PROGRAM P_Demo_DCTIME_TO_STRING
VAR
    // 本程序为 [obsolete] FC / FB 占位演示
    // 新工程统一迁移到 64-bit 等价 FC / FB
END_VAR

// =============================================================================
// Tc2_EtherCAT.DCTIME_TO_STRING 演示程序（[obsolete]）
// =============================================================================
// 场景：维护老工程时偶尔需要查 32-bit DC 时间体系的 helper。本 FC / FB
//       已被 Beckhoff 官方归入 [obsolete]；新工程一律用 64-bit 等价版本。
// 价值：仓库保留本演示与文档，仅供维护老工程时查阅参考。
// 验证步骤：
//   1. 不建议在新工程中使用本 FC / FB
//   2. 若必须使用，参考 PDF 对应章节签名调用
//   3. 优先排期迁移到 64-bit 等价版本
// =============================================================================

// 本 [obsolete] 演示不展示具体调用；请参考 64-bit 版本的 demo 程序
;

END_PROGRAM

(* stored: Version 1.1.0.1, ProductVersion 3.1.4024.5
   POU P_Demo_DCTIME_TO_STRING: Id {417301fd-6078-5fb2-92be-3313c7614fbc}, SpecialFunc None *)
